FUNCTION_BLOCK AxisMovementController
VAR_INPUT
	tolerance: UINT;
	AxisMinus : BOOL;
	AxisPlus: BOOL;
	Control: INT;
	SpeedPWM:INT;
	currentPosition : UINT;
	requiredPosition : UINT;
END_VAR
VAR_OUTPUT
	InPosition:BOOL;
END_VAR
VAR
END_VAR

IF  AboutEqual(
	IN1:= currentPosition,
	IN2:= requiredPosition,
	Tolerance:= tolerance
)
 THEN
	AxisMinus := FALSE;
	AxisPlus := FALSE;
	Control := 0;
	SpeedPWM := 0;
	InPosition := TRUE;
ELSIF currentPosition > requiredPosition AND NOT InPosition THEN
	AxisMinus := TRUE;
	AxisPlus := FALSE;
	Control:= 32;
	SpeedPWM := 5000;
	InPosition := FALSE;
ELSIF currentPosition < requiredPosition AND NOT InPosition THEN
	AxisMinus := FALSE;
	AxisPlus := TRUE;
	Control := 32;
	SpeedPWM := 5000;
	InPosition := FALSE;
ELSE
	AxisMinus := FALSE;
	AxisPlus := FALSE;
	Control := 0;
	SpeedPWM := 0;
	InPosition := FALSE;
END_IF

END_FUNCTION_BLOCK

(* stored: Version 1.1.0.1, ProductVersion 3.1.4024.12
   POU AxisMovementController: Id {156af314-a67a-48d5-b954-455a85c79525}, SpecialFunc None *)
